TYPE ST_ParamActionneur :
STRUCT
	tTimeOut : TIME := T#5S; 					//max time allowed for moving to position bevor xState=TRUE
	xPresenceSensOut : BOOL; 			//If at the out-pos a Sensor is available
	xPresenceSensIn : BOOL; 			//If at the in-pos a Sensor is availaible
	tMoveOutTimeDelay : TIME := T#1S; 	//delay after activating xPresenceSensOut before turning off output. When there is no Sensor, only this time will be used.
	tMoveInTimeDelay : TIME := T#1S; 	//delay after activating xPresenceSensIn before turning off output. When there is no Sensor, only this time will be used.
END_STRUCT
END_TYPE

(* stored: Version 1.1.0.1, ProductVersion 3.1.4020.6
   DUT ST_ParamActionneur: Id {1e55bea4-30da-409a-a73d-7623e8eee451} *)
